# EPICS substitutions: rtApp/Db/tmicro_chan.substitutions
file tmicro_chan.template {
    pattern{M,B,N0,N1,N2,N3,N4,N5,N6,N7,K01,K23,K45,K67}
    {0,0,	0,1,2,3,4,5,6,7,		14,14,14,14}
    {0,1,	8,9,10,11,12,13,14,15,		14,16,16,16}
    {0,2,	16,17,18,19,20,21,22,23,	16,16,16,16}
    {0,3,	24,25,26,27,28,29,30,31,	16,16,16,16}
    {0,4,	32,33,34,35,36,37,38,39,	16,16,16,16}
    {1,0,	64,65,66,67,68,69,70,71,	16,16,16,16}
    {1,1,	72,73,74,75,76,77,78,79,	16,16,16,16}
    {1,2,	80,81,82,83,84,85,86,87,	16,16,16,16}
    {1,3,	88,89,90,91,92,93,94,95,	16,16,16,16}
    {1,4,	96,97,98,99,100,101,102,103,	16,16,18,18}
    {2,0,	128,129,130,131,132,133,134,135,	18,18,18,18}
    {2,1,	136,137,138,139,140,141,142,143,	18,18,18,18}
    {2,2,	144,145,146,147,148,149,150,151,	18,18,18,18}
    {2,3,	152,153,154,155,156,157,158,159,	18,18,18,18}
    {2,4,	160,161,162,163,164,165,166,167,	18,18,18,18}
}
